Staubli VAL3: tskInterlocks.pgx

program tskInterlocks()
  local bool l_bPPSint
  local bool l_bStageint
  local num l_nOldHeartbeat
  local num l_nLastChange
  local string sReturn
  local point LpHere
  local point LpPark
  local num LnDistance
  local num l_nTime
begin
    //header begin
  // PROGRAM tskInterlocks()
  //
  // This pgm is run as a separate task.
  // Will monitor IOC interlocks
  // Utilizes global enable bStopAllMonitor==false set in pgm mnuUtility()
  // Utilizes local enable bEnableMonitor==true set at time of motion command statement, disabled at end of motion
  //
  // Pgm will test for PPS signal while in remote mode.
  // Pgm will test for Z stage position.
  // Pgm will inform IOC of is high level mode.
  //
  // incoming parms:  none
  // outgoing parms:  none
  //
  // called from:  pgm main()
  //
  //
  //  initial release KN
  //header end
  do
    // Turn power off if door is opened and robot in remote mode
    if(nPPS <= 0 and workingMode()==4 and isPowered() )
      logMsg("Door open in remote mode. Power Disconnected")
      popUpMsg("Door open in remote mode. Power Disconnected")
      stopMove()
      resetMotion()
      disablePower()
    endIf

    // Turn off power if robot not at expected z stage position
    if(nStagePos != nStagePosOK and isPowered())
      logMsg("Robot not in correct Z stage position. Power Disconnected")
      popUpMsg("Robot not in correct Z stage position. Power Disconnected")
      stopMove()
      resetMotion()
      disablePower()
    endIf

    if(nHeartbeat !=l_nOldHeartbeat)
      l_nOldHeartbeat = nHeartbeat
      l_nLastChange = clock()
    endIf

    l_nTime = clock()-l_nLastChange

    // Turn off power if robot looses connection to IOC in remote mode
    if(workingMode()==4 and isPowered())
      if(l_nTime>2)
        stopMove()
        resetMotion()
        disablePower()

        logMsg("Lost IOC hearbeat! Power Disconnected")
        sReturn="ERROR 902"
        sReturn=sReturn+": Lost IOC hearbeat! Power Disconnected. "+(toString(".4",l_nTime))
        putln(sReturn)
        logMsg(sReturn)

      endIf
      endIf

    // Report the high level robot mode
    // 0 - Not Parker
    // 1 - Parked
    // 2 - Parked Top

    nRobotMode = 0

    LpHere=here(tSensorTool,world)
    LpPark=jointToPoint(tSensorTool,world,jPark)
    LnDistance=abs(distance(LpHere,LpPark))
    if LnDistance<=nParkTolerance
      nRobotMode = 1
    endIf

    LpHere=here(tSensorTool,world)
    LpPark=jointToPoint(tSensorTool,world,jParkTop)
    LnDistance=abs(distance(LpHere,LpPark))
    if LnDistance<=nParkTolerance
      nRobotMode = 2
    endIf


    delay(0.1)



  until false




end
